PROGRAM MAIN
VAR
	NCI : NCICHannel;
END_VAR

END_PROGRAM

(* stored: Version 1.1.0.1, ProductVersion 3.1.4020.3
   POU MAIN: Id {4b6e6071-00fb-4503-9726-9b98758d323e}, SpecialFunc None *)
